ABB RobotStudio station: Proyecto3_20181222-180958.rsstn

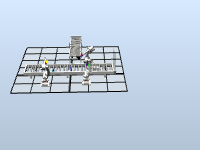
Station Station (saved by RobotStudio 6.6.7701.1025)
Controller System2, task T_ROB1: task frame (RAPID world) sits at (-1000, 1300, 0) mm in the station
Controller Sistema12, task T_ROB1: task frame (RAPID world) sits at (920, -1100, 0) mm, rotated rx 0 ry 0 rz 180 deg in the station
Controller Sistema10, task T_ROB1: task frame (RAPID world) sits at (-920, -900, 0) mm in the station
Controller Sistema10
  mechanical unit ROB_1: JUAN, 6 joints, base frame (0, 0, 0) mm
Controller Sistema12
  mechanical unit ROB_1: ROBERTO, 6 joints, base frame (0, 0, 0) mm
Controller System2
  mechanical unit ROB_1: PACO, 6 joints, base frame (0, 0, 0) mm
Layout (positions relative to the parent item):
  - JUAN [mechanism, from Robots\IRB1600_6_145_G_02.rslib] at (-920, -900, 0) mm; joint values [-0.0712, 0.1084, 0.5172, 0, 0.9452, 3.0704] (rad or m)
  - ROBERTO [mechanism, from Robots\IRB1600_6_145_G_02.rslib] at (920, -1100, 0) mm, rotated rx 0 ry 0 rz 180 deg; joint values [-0.9145, -0.3437, 0.6213, -0.5042, 0.9946, -2.9893] (rad or m)
  - 600_guide [part, from Equipment\Conveyor Guide 600.rslib] at (3800, 50, 0) mm, rotated rx 0 ry 0 rz 180 deg
  - 950_4800_h2 [part, from Equipment\Conveyor 950 4800 h2.rslib] at (475, -2400, 0) mm, rotated rx 0 ry 0 rz 90 deg
  - Pieza_5 [part] at (920, -500, 775) mm
  - Ventosas [smart component]
      signals: DI dedo_Juan, DO Aspira, DI dedo_Roberto, DO Aspira_R
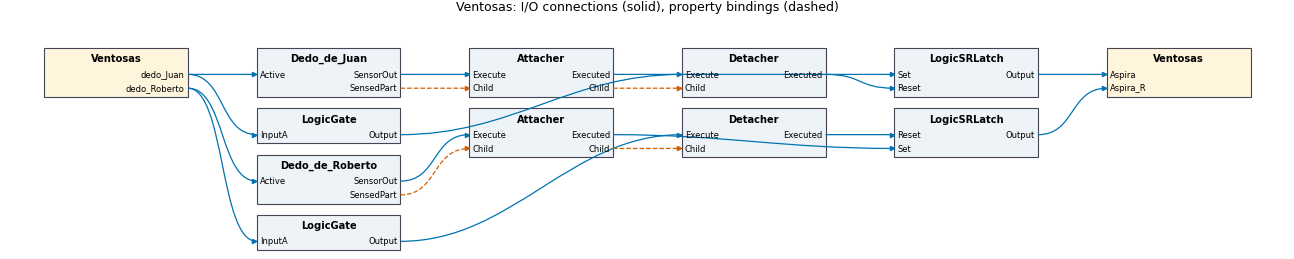
      connections:
        Dedo_de_Juan.SensorOut -> Attacher.Execute
        LogicGate.Output -> Detacher.Execute
        Ventosas.dedo_Juan -> Dedo_de_Juan.Active
        Ventosas.dedo_Juan -> LogicGate.InputA
        Attacher.Executed -> LogicSRLatch.Set
        LogicSRLatch.Output -> Ventosas.Aspira
        Detacher.Executed -> LogicSRLatch.Reset
        Ventosas.dedo_Roberto -> Dedo_de_Roberto.Active
        Dedo_de_Roberto.SensorOut -> Attacher.Execute
        LogicGate.Output -> Detacher.Execute
        Ventosas.dedo_Roberto -> LogicGate.InputA
        Detacher.Executed -> LogicSRLatch.Reset
        Attacher.Executed -> LogicSRLatch.Set
        LogicSRLatch.Output -> Ventosas.Aspira_R
        Dedo_de_Juan.SensedPart => Attacher.Child
        Attacher.Child => Detacher.Child
        Dedo_de_Roberto.SensedPart => Attacher.Child
        Attacher.Child => Detacher.Child
    - Dedo_de_Roberto [smart component, from Components\LineSensor.rslib] at (628.34, -678.2, 925.54) mm, rotated rx 153.61 ry -17.27 rz 135.27 deg
        properties: Start=[0 0 0.08]; End=[0 0 0.11]; Radius=0.002; SensedPart=(none); SensedPoint=[0 0 0]
      - _sensorPart_ [part]
    - Attacher [smart component, from Components\Attacher.rslib]
        properties: Parent=Mano_de_Juan; Flange=0; Child=Pieza_7; Mount=false; Offset=[0 0 0]; Orientation=[0 0 0]
    - LogicGate [smart component, from Components\LogicGate.rslib] at (-1050.67, 0, 0) mm
        properties: Operator=NOT; Delay=0
    - Dedo_de_Juan [smart component, from Components\LineSensor.rslib] at (-209.7, -950.69, 766.04) mm, rotated rx 180 ry 0 rz 0 deg
        properties: Start=[0 0 0.08]; End=[0 0 0.11]; Radius=0.002; SensedPart=Pieza_7; SensedPoint=[-0.177904403686523 -0.95068701171875 0.723270568847656]
      - _sensorPart_ [part]
    - Detacher [smart component, from Components\Detacher.rslib]
        properties: Child=Pieza_7; KeepPosition=true
    - LogicSRLatch [smart component, from Components\LogicSRLatch.rslib]
    - Attacher [smart component, from Components\Attacher.rslib]
        properties: Parent=Mano_de_Roberto; Flange=0; Child=(none); Mount=false; Offset=[0 0 0]; Orientation=[0 0 0]
    - Detacher [smart component, from Components\Detacher.rslib]
        properties: Child=(none); KeepPosition=true
    - LogicSRLatch [smart component, from Components\LogicSRLatch.rslib]
    - LogicGate [smart component, from Components\LogicGate.rslib]
        properties: Operator=NOT; Delay=0
  - Pieza_6 [part] at (370, -1250, 415) mm, rotated rx 0 ry -90 rz 0 deg
  - Cinta_Chasis [smart component]
      signals: DI Montaje_acabado, DO Sensor, DI on, DO SensorP, DO Cinta_on, DO Bandeja_Nueva, DI Pintado, DI rojo, DI azul, DI blanco, DO Sensor_final, DI Sensores_on
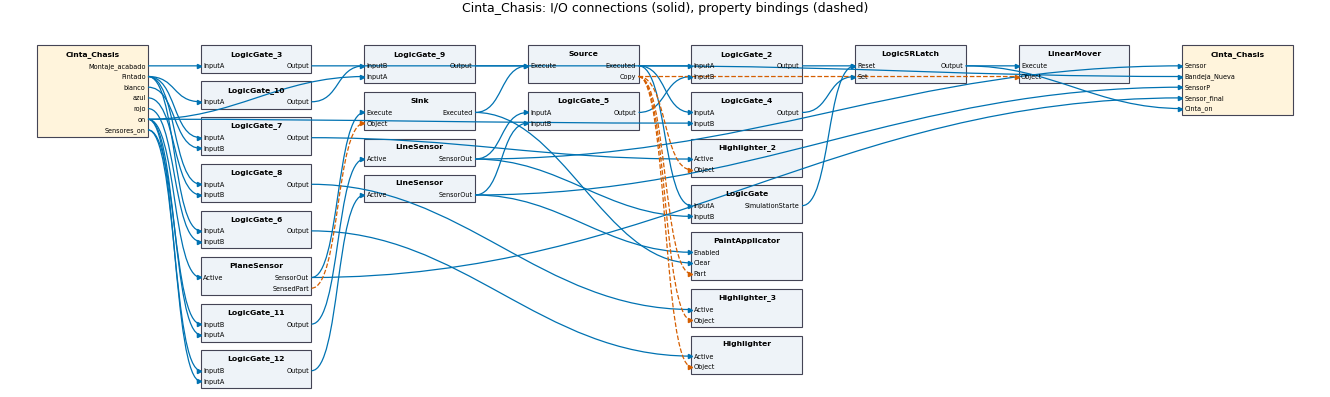
      connections:
        PlaneSensor.SensorOut -> Sink.Execute
        Source.Executed -> LogicGate.InputA
        LineSensor.SensorOut -> LogicGate.InputB
        Cinta_Chasis.Montaje_acabado -> LogicGate_3.InputA
        LogicGate_3.Output -> LogicGate_2.InputA
        LogicGate_2.Output -> LogicSRLatch.Reset
        Source.Executed -> LogicGate_4.InputA
        LogicGate_4.Output -> LogicSRLatch.Set
        LineSensor.SensorOut -> Cinta_Chasis.Sensor
        Sink.Executed -> Source.Execute
        SimulationEvents.SimulationStarted -> LogicSRLatch.Reset
        Source.Executed -> Cinta_Chasis.Bandeja_Nueva
        LineSensor.SensorOut -> Cinta_Chasis.SensorP
        LineSensor.SensorOut -> LogicGate_5.InputA
        LineSensor.SensorOut -> LogicGate_5.InputB
        LogicGate_5.Output -> LogicGate_2.InputB
        Cinta_Chasis.Pintado -> LogicGate_6.InputA
        Cinta_Chasis.Pintado -> LogicGate_8.InputA
        Cinta_Chasis.Pintado -> LogicGate_7.InputA
        Cinta_Chasis.blanco -> LogicGate_7.InputB
        Cinta_Chasis.azul -> LogicGate_8.InputB
        Cinta_Chasis.rojo -> LogicGate_6.InputB
        LogicGate_7.Output -> Highlighter_2.Active
        LogicGate_8.Output -> Highlighter_3.Active
        LogicGate_6.Output -> Highlighter.Active
        LineSensor.SensorOut -> PaintApplicator.Enabled
        Sink.Executed -> PaintApplicator.Clear
        Cinta_Chasis.Pintado -> LogicGate_10.InputA
        LogicGate_10.Output -> LogicGate_9.InputB
        LogicGate_9.Output -> Source.Execute
        Cinta_Chasis.on -> LogicGate_9.InputA
        PlaneSensor.SensorOut -> Cinta_Chasis.Sensor_final
        Cinta_Chasis.on -> PlaneSensor.Active
        Cinta_Chasis.Sensores_on -> LogicGate_11.InputB
        Cinta_Chasis.on -> LogicGate_11.InputA
        LogicGate_11.Output -> LineSensor.Active
        Cinta_Chasis.Sensores_on -> LogicGate_12.InputB
        Cinta_Chasis.on -> LogicGate_12.InputA
        LogicGate_12.Output -> LineSensor.Active
        Cinta_Chasis.on -> LogicGate_4.InputB
        LogicSRLatch.Output -> Cinta_Chasis.Cinta_on
        LogicSRLatch.Output -> LinearMover.Execute
        PlaneSensor.SensedPart => Sink.Object
        Source.Copy => LinearMover.Object
        Source.Copy => Highlighter.Object
        Source.Copy => Highlighter_3.Object
        Source.Copy => Highlighter_2.Object
        Source.Copy => PaintApplicator.Part
    - Source [smart component, from Components\Source.rslib] at (0, 0, 0) mm
        properties: Source=Chasis; Copy=(none); Parent=(none); Position=[-0.2 2.75 0.6]; Orientation=[0 3.14159265358979 -1.5707963267949]; Transient=false; PhysicsBehavior=0
    - PlaneSensor [smart component, from Components\PlaneSensor.rslib]
        properties: Origin=[-0.52 -2.42 0.45]; Axis1=[0 0 1]; Axis2=[1.05 0 0]; SensedPart=(none)
      - _sensorPart_ [part]
    - Sink [smart component, from Components\Sink.rslib]
        properties: Object=(none)
    - LinearMover [smart component, from Components\LinearMover.rslib]
        properties: Object=(none); Direction=[0 -0.001 0]; Speed=0.5; Reference=Global; ReferenceObject=(none)
    - LineSensor [smart component, from Components\LineSensor.rslib]
        properties: Start=[0.040738 -1.264377 0.404542]; End=[0.040738 -1.264377 0.44]; Radius=0.005; SensedPart=(none); SensedPoint=[0 0 0]
      - _sensorPart_ [part]
    - LogicSRLatch [smart component, from Components\LogicSRLatch.rslib]
    - LogicGate_2 [smart component, from Components\LogicGate.rslib]
        properties: Operator=AND; Delay=0
    - LogicGate_3 [smart component, from Components\LogicGate.rslib]
        properties: Operator=NOT; Delay=0
    - LogicGate_4 [smart component, from Components\LogicGate.rslib]
        properties: Operator=OR; Delay=0
    - LineSensor [smart component, from Components\LineSensor.rslib]
        properties: Start=[0.04074 0.99 0.404]; End=[0.04074 0.99 0.44]; Radius=0.005; SensedPart=(none); SensedPoint=[0 0 0]
      - _sensorPart_ [part]
    - LogicGate_5 [smart component, from Components\LogicGate.rslib]
        properties: Operator=OR; Delay=0
    - Highlighter [smart component, from Components\Highlighter.rslib]
        properties: Object=(none); Color=[255 0 0]; Opacity=255
    - Highlighter_2 [smart component, from Components\Highlighter.rslib]
        properties: Object=(none); Color=[255 255 255]; Opacity=255
    - Highlighter_3 [smart component, from Components\Highlighter.rslib]
        properties: Object=(none); Color=[0 0 255]; Opacity=255
    - LogicGate_6 [smart component, from Components\LogicGate.rslib]
        properties: Operator=AND; Delay=0
    - LogicGate_7 [smart component, from Components\LogicGate.rslib]
        properties: Operator=AND; Delay=0
    - LogicGate_8 [smart component, from Components\LogicGate.rslib]
        properties: Operator=AND; Delay=0
    - PaintApplicator [smart component, from Components\PaintApplicator.rslib] at (-273.7, 1300, 862.91) mm, rotated rx 180 ry 9.88 rz 180 deg
        properties: Part=(none); Color=-1; ShowPreviewCone=true; Strength=0.025; Range=0.5; Width=0.5; Height=0.5
    - LogicGate_9 [smart component, from Components\LogicGate.rslib]
        properties: Operator=AND; Delay=0
    - LogicGate_10 [smart component, from Components\LogicGate.rslib]
        properties: Operator=NOT; Delay=0
    - LogicGate_11 [smart component, from Components\LogicGate.rslib]
        properties: Operator=AND; Delay=0
    - LogicGate_12 [smart component, from Components\LogicGate.rslib]
        properties: Operator=AND; Delay=0
  - Mano_de_Juan [mechanism] at (-209.7, -950.69, 766.04) mm, rotated rx 180 ry 0 rz 0 deg
      TCP Mano_de_Juan at (0, 0, 100) mm
      links: Pieza_7
  - rueda_atras_azul [part] at (1106.02, -365.17, 900) mm, rotated rx 180 ry 0 rz 0 deg
  - rueda_atras_azul_2 [part] at (1107.91, -123.11, 900) mm, rotated rx 180 ry 0 rz 0 deg
  - rueda_delante_azul [part] at (1451.59, -315.99, 875) mm, rotated rx 90 ry 0 rz 0 deg
  - arandela [part] at (1451.94, -129.36, 875) mm, rotated rx 90 ry 0 rz 0 deg
  - Mano_de_Roberto [mechanism] at (628.34, -678.2, 925.54) mm, rotated rx 153.61 ry -17.27 rz 135.27 deg
      TCP Mano_de_Roberto at (0, 0, 100) mm
      links: Pieza_7
  - PACO [mechanism, from Robots\IRB1600_6_145_G_02.rslib] at (-1000, 1300, 0) mm; joint values [0, -0.5373, 0.3681, 0, 0.6599, 0] (rad or m)
  - Binzel_air_22 [mechanism, from Tools\Binzel_air_22.rslib] at (-559.51, 1300, 1158.26) mm, rotated rx 180 ry 61.88 rz 180 deg
  - Bandeja_Chasis [smart component]
      signals: DI Cinta_on, DI Montaje_acabado, DI Bandeja_nueva, DO Sensor_final
      connections:
        PlaneSensor_2.SensorOut -> Sink.Execute
        Bandeja_Chasis.Bandeja_nueva -> Source.Execute
        LogicGate_13.Output -> PlaneSensor_2.Active
        Bandeja_Chasis.Cinta_on -> LogicGate_13.InputA
        LogicSRLatch.Output -> LinearMover.Execute
        Source.Executed -> LogicSRLatch.Set
        Bandeja_Chasis.Cinta_on -> LinearMover.Execute
        LogicGate_14.Output -> PlaneSensor_2.Active
        Bandeja_Chasis.Montaje_acabado -> LogicGate_14.InputB
        Bandeja_Chasis.Cinta_on -> LogicGate_14.InputA
        PlaneSensor_2.SensedPart => Sink.Object
        Source.Copy => LinearMover.Object
    - Source [smart component, from Components\Source.rslib]
        properties: Source=Bandeja; Copy=(none); Parent=(none); Position=[0 2.5 0]; Orientation=[0 0 0]; Transient=false; PhysicsBehavior=0
    - Sink [smart component, from Components\Sink.rslib]
        properties: Object=(none)
    - LinearMover [smart component, from Components\LinearMover.rslib]
        properties: Object=(none); Direction=[0 -0.001 0]; Speed=0.5; Reference=Global; ReferenceObject=(none)
    - PlaneSensor_2 [smart component, from Components\PlaneSensor.rslib]
        properties: Origin=[-0.52 -2.5 0.35]; Axis1=[0 0 1]; Axis2=[1.05 0 0]; SensedPart=(none)
      - _sensorPart_ [part]
    - LogicGate_14 [smart component, from Components\LogicGate.rslib]
        properties: Operator=OR; Delay=0
  - Bandeja [part]
  - Chasis [part] at (-200, -1494, 610) mm, rotated rx 180 ry 0 rz 90 deg
  - LogicGate_9 [smart component, from Components\LogicGate.rslib]
      properties: Operator=AND; Delay=0
  - LogicGate_10 [smart component, from Components\LogicGate.rslib]
      properties: Operator=NOT; Delay=0
  - rueda_atras_blanca [part] at (1106.02, -365.17, 900) mm, rotated rx 180 ry 0 rz 0 deg
  - rueda_atras_blanca_2 [part] at (1107.91, -123.11, 900) mm, rotated rx 180 ry 0 rz 0 deg
  - rueda_delante_blanca [part] at (1451.59, -315.99, 875) mm, rotated rx 90 ry 0 rz 0 deg
  - rueda_atras_roja [part] at (1106.02, -365.17, 900) mm, rotated rx 180 ry 0 rz 0 deg
  - rueda_atras_roja_2 [part] at (1107.91, -123.11, 900) mm, rotated rx 180 ry 0 rz 0 deg
  - rueda_delante_roja [part] at (1451.59, -315.99, 875) mm, rotated rx 90 ry 0 rz 0 deg
  - Componente inteligente_1 [smart component]
      signals: DI Piezas_cogidas, DO piezas_mov, DI Piezas_colocadas
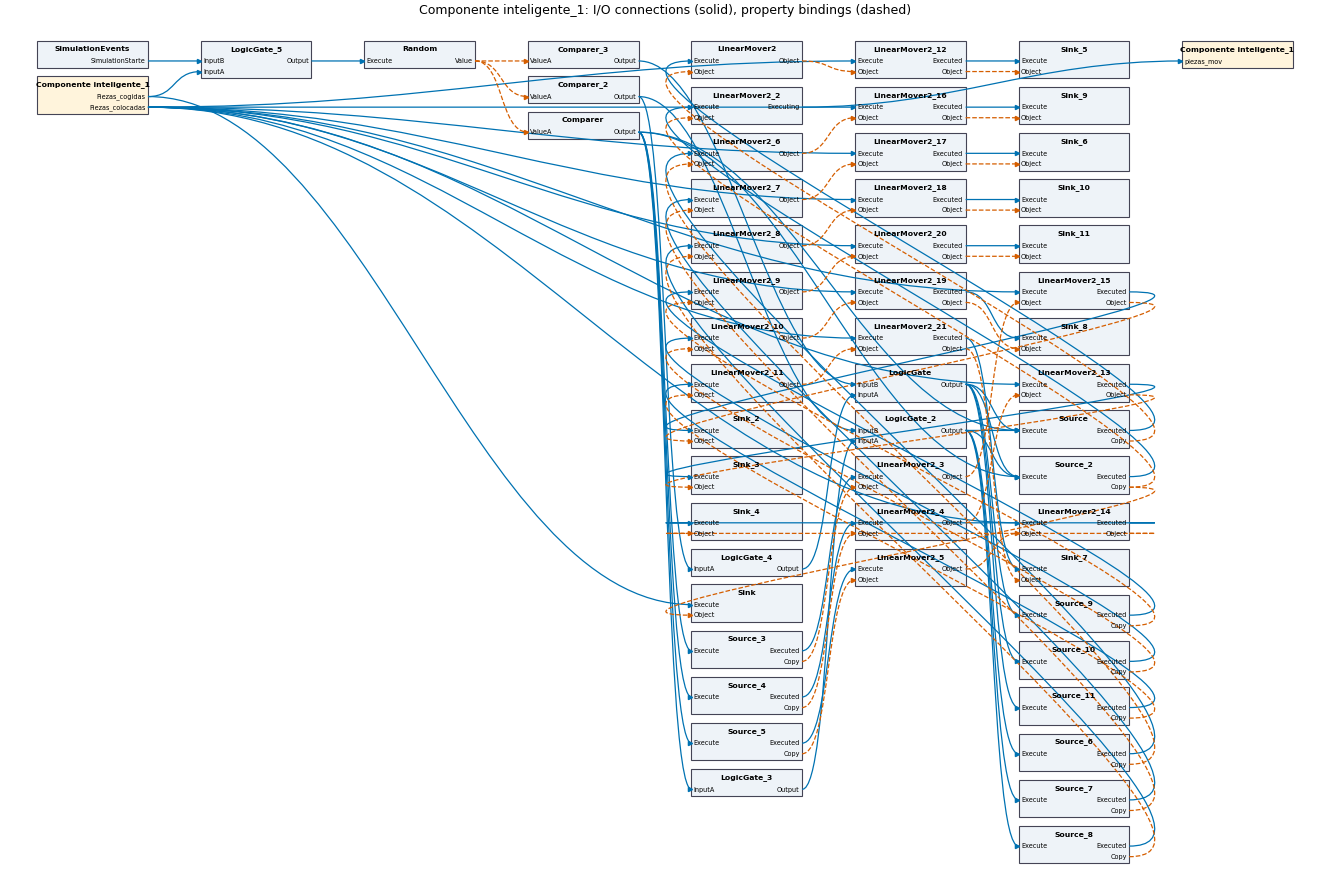
      connections:
        Comparer_3.Output -> LogicGate.InputB
        Comparer_2.Output -> LogicGate_2.InputB
        Comparer.Output -> Source.Execute
        Comparer.Output -> Source_2.Execute
        Comparer.Output -> Source_3.Execute
        Comparer.Output -> Source_4.Execute
        Comparer.Output -> Source_5.Execute
        Comparer.Output -> LogicGate_3.InputA
        LogicGate_3.Output -> LogicGate_2.InputA
        LogicGate_2.Output -> Source_6.Execute
        LogicGate_2.Output -> Source_7.Execute
        LogicGate_2.Output -> Source_8.Execute
        LogicGate_2.Output -> Source_2.Execute
        LogicGate_2.Output -> Source.Execute
        Comparer_2.Output -> LogicGate_4.InputA
        LogicGate_4.Output -> LogicGate.InputA
        LogicGate.Output -> Source_9.Execute
        LogicGate.Output -> Source_10.Execute
        LogicGate.Output -> Source_11.Execute
        LogicGate.Output -> Source_2.Execute
        LogicGate.Output -> Source.Execute
        Source.Executed -> LinearMover2.Execute
        Source_2.Executed -> LinearMover2_2.Execute
        Source_3.Executed -> LinearMover2_3.Execute
        Source_4.Executed -> LinearMover2_4.Execute
        Source_5.Executed -> LinearMover2_5.Execute
        Source_6.Executed -> LinearMover2_6.Execute
        Source_7.Executed -> LinearMover2_7.Execute
        Source_8.Executed -> LinearMover2_8.Execute
        Source_9.Executed -> LinearMover2_9.Execute
        Source_10.Executed -> LinearMover2_10.Execute
        Source_11.Executed -> LinearMover2_11.Execute
        SimulationEvents.SimulationStarted -> LogicGate_5.InputB
        Componente inteligente_1.Piezas_cogidas -> LogicGate_5.InputA
        LogicGate_5.Output -> Random.Execute
        Componente inteligente_1.Piezas_cogidas -> Sink.Execute
        LinearMover2_2.Executing -> Componente inteligente_1.piezas_mov
        Componente inteligente_1.Piezas_colocadas -> LinearMover2_15.Execute
        Componente inteligente_1.Piezas_colocadas -> LinearMover2_13.Execute
        Componente inteligente_1.Piezas_colocadas -> LinearMover2_14.Execute
        Componente inteligente_1.Piezas_colocadas -> LinearMover2_12.Execute
        Componente inteligente_1.Piezas_colocadas -> LinearMover2_16.Execute
        Componente inteligente_1.Piezas_colocadas -> LinearMover2_17.Execute
        Componente inteligente_1.Piezas_colocadas -> LinearMover2_18.Execute
        Componente inteligente_1.Piezas_colocadas -> LinearMover2_20.Execute
        Componente inteligente_1.Piezas_colocadas -> LinearMover2_19.Execute
        Componente inteligente_1.Piezas_colocadas -> LinearMover2_21.Execute
        LinearMover2_15.Executed -> Sink_2.Execute
        LinearMover2_13.Executed -> Sink_3.Execute
        LinearMover2_14.Executed -> Sink_4.Execute
        LinearMover2_12.Executed -> Sink_5.Execute
        LinearMover2_16.Executed -> Sink_9.Execute
        LinearMover2_17.Executed -> Sink_6.Execute
        LinearMover2_18.Executed -> Sink_10.Execute
        LinearMover2_20.Executed -> Sink_11.Execute
        LinearMover2_19.Executed -> Sink_8.Execute
        LinearMover2_21.Executed -> Sink_7.Execute
        Random.Value => Comparer.ValueA
        Random.Value => Comparer_2.ValueA
        Random.Value => Comparer_3.ValueA
        Source.Copy => LinearMover2.Object
        Source_2.Copy => LinearMover2_2.Object
        Source_3.Copy => LinearMover2_3.Object
        Source_4.Copy => LinearMover2_4.Object
        Source_5.Copy => LinearMover2_5.Object
        Source_6.Copy => LinearMover2_6.Object
        Source_7.Copy => LinearMover2_7.Object
        Source_8.Copy => LinearMover2_8.Object
        Source_9.Copy => LinearMover2_9.Object
        Source_10.Copy => LinearMover2_10.Object
        Source_11.Copy => LinearMover2_11.Object
        Source_2.Copy => Sink.Object
        LinearMover2.Object => LinearMover2_12.Object
        LinearMover2_3.Object => LinearMover2_15.Object
        LinearMover2_4.Object => LinearMover2_13.Object
        LinearMover2_5.Object => LinearMover2_14.Object
        LinearMover2_6.Object => LinearMover2_16.Object
        LinearMover2_7.Object => LinearMover2_17.Object
        LinearMover2_8.Object => LinearMover2_18.Object
        LinearMover2_9.Object => LinearMover2_20.Object
        LinearMover2_10.Object => LinearMover2_19.Object
        LinearMover2_11.Object => LinearMover2_21.Object
        LinearMover2_15.Object => Sink_2.Object
        LinearMover2_13.Object => Sink_3.Object
        LinearMover2_14.Object => Sink_4.Object
        LinearMover2_12.Object => Sink_5.Object
        LinearMover2_16.Object => Sink_9.Object
        LinearMover2_17.Object => Sink_6.Object
        LinearMover2_18.Object => Sink_10.Object
        LinearMover2_20.Object => Sink_11.Object
        LinearMover2_19.Object => Sink_8.Object
        LinearMover2_21.Object => Sink_7.Object
    - LogicGate [smart component, from Components\LogicGate.rslib]
        properties: Operator=AND; Delay=0
    - SimulationEvents [smart component, from Components\SimulationEvents.rslib]
    - Comparer [smart component, from Components\Comparer.rslib]
        properties: ValueA=0.882498855647863; Operator=<=; ValueB=1
    - Comparer_2 [smart component, from Components\Comparer.rslib]
        properties: ValueA=0.882498855647863; Operator=<=; ValueB=2
    - Comparer_3 [smart component, from Components\Comparer.rslib]
        properties: ValueA=0.882498855647863; Operator=<=; ValueB=3
    - Random [smart component, from Components\Random.rslib]
        properties: Value=0.882498855647863; Min=0; Max=3
    - LogicGate_2 [smart component, from Components\LogicGate.rslib]
        properties: Operator=AND; Delay=0
    - Source [smart component, from Components\Source.rslib]
        properties: Source=arandela; Copy=(none); Parent=(none); Position=[3.451939 -0.129363 0.875]; Orientation=[1.5707963267949 0 0]; Transient=false; PhysicsBehavior=0
    - Source_2 [smart component, from Components\Source.rslib]
        properties: Source=Pieza_5; Copy=(none); Parent=(none); Position=[2.92 -0.5 0.775]; Orientation=[0 0 0]; Transient=false; PhysicsBehavior=0
    - Source_3 [smart component, from Components\Source.rslib]
        properties: Source=rueda_atras_azul; Copy=(none); Parent=(none); Position=[3.107912 -0.123105 0.9]; Orientation=[3.14159265358979 0 0]; Transient=false; PhysicsBehavior=0
    - Source_4 [smart component, from Components\Source.rslib]
        properties: Source=rueda_atras_azul_2; Copy=(none); Parent=(none); Position=[3.106016 -0.365172 0.9]; Orientation=[3.14159265358979 0 0]; Transient=false; PhysicsBehavior=0
    - Source_5 [smart component, from Components\Source.rslib]
        properties: Source=rueda_delante_azul; Copy=(none); Parent=(none); Position=[3.451589 -0.315989 0.875]; Orientation=[1.5707963267949 0 0]; Transient=false; PhysicsBehavior=0
    - Source_6 [smart component, from Components\Source.rslib]
        properties: Source=rueda_atras_roja; Copy=(none); Parent=(none); Position=[3.107912 -0.123105 0.9]; Orientation=[3.14159265358979 0 0]; Transient=false; PhysicsBehavior=0
    - Source_7 [smart component, from Components\Source.rslib]
        properties: Source=rueda_atras_roja_2; Copy=(none); Parent=(none); Position=[3.106016 -0.365172 0.9]; Orientation=[3.14159265358979 0 0]; Transient=false; PhysicsBehavior=0
    - Source_8 [smart component, from Components\Source.rslib]
        properties: Source=rueda_delante_roja; Copy=(none); Parent=(none); Position=[3.451589 -0.315989 0.875]; Orientation=[1.5707963267949 0 0]; Transient=false; PhysicsBehavior=0
    - Source_9 [smart component, from Components\Source.rslib]
        properties: Source=rueda_atras_blanca; Copy=(none); Parent=(none); Position=[3.107912 -0.123105 0.9]; Orientation=[3.14159265358979 0 0]; Transient=false; PhysicsBehavior=0
    - Source_10 [smart component, from Components\Source.rslib]
        properties: Source=rueda_atras_blanca_2; Copy=(none); Parent=(none); Position=[3.106016 -0.365172 0.9]; Orientation=[3.14159265358979 0 0]; Transient=false; PhysicsBehavior=0
    - Source_11 [smart component, from Components\Source.rslib]
        properties: Source=rueda_delante_blanca; Copy=(none); Parent=(none); Position=[3.451589 -0.315989 0.875]; Orientation=[1.5707963267949 0 0]; Transient=false; PhysicsBehavior=0
    - LogicGate_3 [smart component, from Components\LogicGate.rslib]
        properties: Operator=NOT; Delay=0
    - LogicGate_4 [smart component, from Components\LogicGate.rslib]
        properties: Operator=NOT; Delay=0
    - LinearMover2 [smart component, from Components\LinearMover2.rslib]
        properties: Object=(none); Direction=[-1 0 0]; Distance=2; Duration=4; Reference=Global; ReferenceObject=(none)
    - LinearMover2_2 [smart component, from Components\LinearMover2.rslib]
        properties: Object=(none); Direction=[-1 0 0]; Distance=2; Duration=4; Reference=Global; ReferenceObject=(none)
    - LinearMover2_3 [smart component, from Components\LinearMover2.rslib]
        properties: Object=(none); Direction=[-1 0 0]; Distance=2; Duration=4; Reference=Global; ReferenceObject=(none)
    - LinearMover2_4 [smart component, from Components\LinearMover2.rslib]
        properties: Object=(none); Direction=[-1 0 0]; Distance=2; Duration=4; Reference=Global; ReferenceObject=(none)
    - LinearMover2_5 [smart component, from Components\LinearMover2.rslib]
        properties: Object=(none); Direction=[-1 0 0]; Distance=2; Duration=4; Reference=Global; ReferenceObject=(none)
    - LinearMover2_6 [smart component, from Components\LinearMover2.rslib]
        properties: Object=(none); Direction=[-1 0 0]; Distance=2; Duration=4; Reference=Global; ReferenceObject=(none)
    - LinearMover2_7 [smart component, from Components\LinearMover2.rslib]
        properties: Object=(none); Direction=[-1 0 0]; Distance=2; Duration=4; Reference=Global; ReferenceObject=(none)
    - LinearMover2_8 [smart component, from Components\LinearMover2.rslib]
        properties: Object=(none); Direction=[-1 0 0]; Distance=2; Duration=4; Reference=Global; ReferenceObject=(none)
    - LinearMover2_9 [smart component, from Components\LinearMover2.rslib]
        properties: Object=(none); Direction=[-1 0 0]; Distance=2; Duration=4; Reference=Global; ReferenceObject=(none)
    - LinearMover2_10 [smart component, from Components\LinearMover2.rslib]
        properties: Object=(none); Direction=[-1 0 0]; Distance=2; Duration=4; Reference=Global; ReferenceObject=(none)
    - LinearMover2_11 [smart component, from Components\LinearMover2.rslib]
        properties: Object=(none); Direction=[-1 0 0]; Distance=2; Duration=4; Reference=Global; ReferenceObject=(none)
    - LogicGate_5 [smart component, from Components\LogicGate.rslib]
        properties: Operator=OR; Delay=0
    - Sink [smart component, from Components\Sink.rslib]
        properties: Object=(none)
    - LinearMover2_12 [smart component, from Components\LinearMover2.rslib]
        properties: Object=(none); Direction=[0 -0.001 0]; Distance=2; Duration=4; Reference=Global; ReferenceObject=(none)
    - LinearMover2_13 [smart component, from Components\LinearMover2.rslib]
        properties: Object=(none); Direction=[0 -0.001 0]; Distance=2; Duration=4; Reference=Global; ReferenceObject=(none)
    - LinearMover2_14 [smart component, from Components\LinearMover2.rslib]
        properties: Object=(none); Direction=[0 -0.001 0]; Distance=2; Duration=4; Reference=Global; ReferenceObject=(none)
    - LinearMover2_15 [smart component, from Components\LinearMover2.rslib]
        properties: Object=(none); Direction=[0 -0.001 0]; Distance=2; Duration=4; Reference=Global; ReferenceObject=(none)
    - LinearMover2_16 [smart component, from Components\LinearMover2.rslib]
        properties: Object=(none); Direction=[0 -0.001 0]; Distance=2; Duration=4; Reference=Global; ReferenceObject=(none)
    - LinearMover2_17 [smart component, from Components\LinearMover2.rslib]
        properties: Object=(none); Direction=[0 -0.001 0]; Distance=2; Duration=4; Reference=Global; ReferenceObject=(none)
    - LinearMover2_18 [smart component, from Components\LinearMover2.rslib]
        properties: Object=(none); Direction=[1 0 0]; Distance=0; Duration=0; Reference=Global; ReferenceObject=(none)
    - LinearMover2_19 [smart component, from Components\LinearMover2.rslib]
        properties: Object=(none); Direction=[0 -0.001 0]; Distance=2; Duration=4; Reference=Global; ReferenceObject=(none)
    - LinearMover2_20 [smart component, from Components\LinearMover2.rslib]
        properties: Object=(none); Direction=[0 -0.001 0]; Distance=2; Duration=4; Reference=Global; ReferenceObject=(none)
    - LinearMover2_21 [smart component, from Components\LinearMover2.rslib]
        properties: Object=(none); Direction=[0 -0.001 0]; Distance=2; Duration=4; Reference=Global; ReferenceObject=(none)
    - Sink_2 [smart component, from Components\Sink.rslib]
        properties: Object=(none)
    - Sink_3 [smart component, from Components\Sink.rslib]
        properties: Object=(none)
    - Sink_4 [smart component, from Components\Sink.rslib]
        properties: Object=(none)
    - Sink_5 [smart component, from Components\Sink.rslib]
        properties: Object=(none)
    - Sink_6 [smart component, from Components\Sink.rslib]
        properties: Object=(none)
    - Sink_7 [smart component, from Components\Sink.rslib]
        properties: Object=(none)
    - Sink_8 [smart component, from Components\Sink.rslib]
        properties: Object=(none)
    - Sink_9 [smart component, from Components\Sink.rslib]
        properties: Object=(none)
    - Sink_10 [smart component, from Components\Sink.rslib]
        properties: Object=(none)
    - Sink_11 [smart component, from Components\Sink.rslib]
        properties: Object=(none)
Attachment: Dedo_de_Roberto is attached to Mano_de_Roberto / Pieza_7
Attachment: Dedo_de_Juan is attached to Mano_de_Juan / Pieza_7
Attachment: Source is attached to Mano_de_Roberto / Pieza_7
Attachment: PaintApplicator is attached to Binzel_air_22 / Binzel_air_22_sat
Attachment: Mano_de_Juan is attached to JUAN / Link6
Attachment: Mano_de_Roberto is attached to ROBERTO / Link6
Attachment: Binzel_air_22 is attached to PACO / Link6
Attachment: Componente inteligente_1 is attached to ROBERTO / Link6
Station logic (signal -> signal, property => property):
  Ventosas.Aspira -> Sistema10.PiezaCogida_Juan
  Sistema10.ActivaMano_Juan -> Ventosas.dedo_Juan
  Cinta_Chasis.Sensor -> Sistema10.Sensor_cinta
  Sistema10.Montaje_fin -> Cinta_Chasis.Montaje_acabado
  Sistema12.ActivaMano_Roberto -> Ventosas.dedo_Roberto
  Ventosas.Aspira_R -> Sistema12.PiezaCogida_Roberto
  Sistema10.Montaje_fin -> Bandeja_Chasis.Montaje_acabado
  Cinta_Chasis.SensorP -> System2.Sensor
  System2.Pintado -> Cinta_Chasis.Pintado
  Sistema10.Cinta_on -> LogicGate_9.InputA
  LogicGate_10.Output -> LogicGate_9.InputB
  System2.Apaga_Cinta -> LogicGate_10.InputA
  LogicGate_9.Output -> Cinta_Chasis.on
  Cinta_Chasis.Sensor_final -> System2.Sensor_final
  Sistema10.Sensores -> Cinta_Chasis.Sensores_on
  Cinta_Chasis.Bandeja_Nueva -> Bandeja_Chasis.Bandeja_nueva
  Cinta_Chasis.Cinta_on -> Bandeja_Chasis.Cinta_on
  Bandeja_Chasis.Sensor_final -> Sistema10.Sensor_final
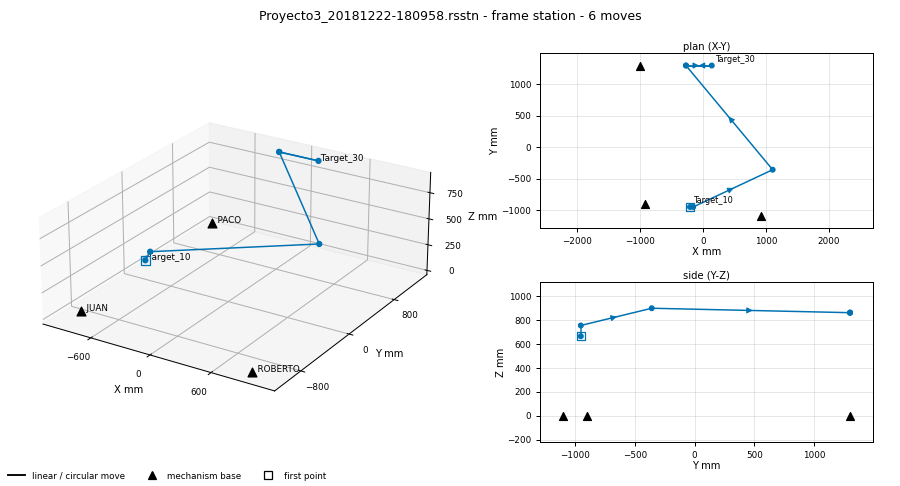
[picture p0: tool path of Proyecto3_20181222-180958.rsstn in frame station, 6 of 6 moves have a stored position in this frame; points joined in program order, loops and branches not executed]
Targets, tools, work objects and paths stored in the station, written as RAPID:
! task T_ROB1
MODULE Module1
  CONST robtarget Target_10:=[[710.302,-50.687,666.042],[0,1,0,0],[-1,0,1,0],[9E+09,9E+09,9E+09,9E+09,9E+09,9E+09]];
  CONST robtarget Target_20:=[[760.301980587,-50.686989693,756.042035513],[-0.000000033,1,-0.000000027,0.000000018],[-1,-1,1,0],[9E+09,9E+09,9E+09,9E+09,9E+09,9E+09]];
  PROC Path_10()
    MoveL Target_10,v1000,z100,Mano_de_Juan\WObj:=wobj0;
    SetDO ActivaMano_Juan,1;
    MoveL Target_20,v1000,z100,Mano_de_Juan\WObj:=wobj0;
  ENDPROC
ENDMODULE

! task T_ROB1
MODULE CalibData
  PERS tooldata Mano_de_Juan:=[TRUE,[[0,0,100],[1,0,0,0]],[1,[0,0,1],[1,0,0,0],0,0,0]];
ENDMODULE

! task T_ROB1
MODULE CalibData
  PERS tooldata Mano_de_Roberto:=[TRUE,[[0,0,100],[1,0,0,0]],[1,[0,0,1],[1,0,0,0],0,0,0]];
ENDMODULE

! task T_ROB1
MODULE Module1
  CONST robtarget Target_10:=[[-185.627,-742.177,900],[0,0,0,1],[0,0,0,0],[9E+09,9E+09,9E+09,9E+09,9E+09,9E+09]];
  PROC Path_10()
    MoveL Target_10,v1000,z100,Mano_de_Roberto\WObj:=wobj0;
  ENDPROC
ENDMODULE

! task T_ROB1
MODULE CalibData
  PERS tooldata tWeldGun:=[TRUE,[[125.800591275,0,391.268161315],[0.898794046,0,0.438371147,0]],[3,[0,0,100],[0,1,0,0],0,0,0]];
  TASK PERS wobjdata Workobject_1:=[FALSE,TRUE,"",[[550,-400,440],[1,0,0,0]],[[0,0,0],[1,0,0,0]]];
ENDMODULE

! task T_ROB1
MODULE Module1
  CONST robtarget Target_10:=[[441.621481043,0,1158.262985958],[0.514156313,0,0.8576965,0],[0,0,0,0],[9E+09,9E+09,9E+09,9E+09,9E+09,9E+09]];
  CONST robtarget Target_20:=[[176.295674853,400,422.909917876],[0.086131219,0,0.996283801,0],[0,0,0,0],[9E+09,9E+09,9E+09,9E+09,9E+09,9E+09]];
  CONST robtarget Target_30:=[[586.583995183,400,422.909955081],[0.086131256,0,0.996283798,0],[0,0,0,0],[9E+09,9E+09,9E+09,9E+09,9E+09,9E+09]];
  PROC Path_10()
    MoveL Target_20,v1000,fine,tWeldGun\WObj:=Workobject_1;
    MoveL Target_30,v1000,fine,tWeldGun\WObj:=Workobject_1;
    MoveL Target_20,v1000,fine,tWeldGun\WObj:=Workobject_1;
  ENDPROC
  PROC Inicio()
    SetDO Apaga_Cinta,1;
    SetDO Apaga_Cinta,0;
    SetDO Pintado,1;
    SetDO Pintado,0;
  ENDPROC
  PROC main()
    SetDO Apaga_Cinta,0;
    Inicio;
    WaitDI Sensor,1;
    SetDO Apaga_Cinta,1;
    Path_10;
    WaitTime 0.2;
    SetDO Pintado,1;
    WaitTime 0.2;
    SetDO Apaga_Cinta,0;
    WaitDI Sensor_final,1;
    WaitTime 2;
    SetDO Pintado,0;
  ENDPROC
ENDMODULE

